FUNCTION TryConvert_DINT_TO_DT : BOOL
VAR_INPUT
	in : DINT;
	out : REFERENCE TO DT;
END_VAR

IF in < DatatypeLimits.MIN_VALUE_OF_DINT_WHICH_CAN_BE_HELD_IN_A_DT THEN
	RETURN;
END_IF

out := DINT_TO_DT(in);
TryConvert_DINT_TO_DT := TRUE;

END_FUNCTION

(* stored: Version 1.1.0.1, ProductVersion 3.1.4024.12
   POU TryConvert_DINT_TO_DT: Id {ea94dd40-f625-4d8f-bf9e-c37dfac33480}, SpecialFunc None *)
